PROGRAM MAIN
VAR
END_VAR

PRG_Testing();

END_PROGRAM

(* stored: Version 1.1.0.1, ProductVersion 3.1.4024.12
   POU MAIN: Id {8c54dcfa-95ea-4b9a-a141-36f7e978e526}, SpecialFunc None *)
